INTERFACE I_QuantityLREALPublic EXTENDS I_QuantityPublic, I_QuantityLREAL


METHOD Copy
VAR_INPUT
    QuantityToCopy : I_QuantityLREAL;
END_VAR
END_METHOD


PROPERTY Val : LREAL
SET
END_SET
END_PROPERTY

END_INTERFACE

(* stored: Version 1.1.0.1
   Itf I_QuantityLREALPublic: Id {054488e9-23a0-4927-be35-da45401b7565}
   Method Copy: Id {74285296-16ea-43e3-bcb3-6f7ad2de0fcf}
   Property Val: Id {7bcda038-7fd6-4d42-9931-f7f5c952fa96}
   Set Set: Id {6193ebdc-af3c-429e-84f0-fe7b372da9c3} *)
